{attribute 'linkalways'} 
{attribute 'no_explicit_call' := 'This FB is a CLASS and must be accessed using methods or properties'}
{attribute 'enable_dynamic_creation'}
FUNCTION_BLOCK Node_F_VN_InsertIntoContainer_SINT EXTENDS VisionNode
VAR
    nElement : _SINT(0);
    ipContainer : _ITcVnContainer;
    nIndex : _ULINT(0);
    hrPrev : _HRESULT(S_OK);
    hresult : _HRESULT(S_OK);
END_VAR

METHOD PUBLIC  Clone : I_Node
VAR
	pNode : POINTER TO Node_F_VN_InsertIntoContainer_SINT;
END_VAR
pNode := __NEW(Node_F_VN_InsertIntoContainer_SINT);
Clone := pNode^;
END_METHOD

METHOD FB_init : BOOL
VAR_INPUT
	bInitRetains : BOOL; // if TRUE, the retain variables are initialized (warm start / cold start)
	bInCopyCode : BOOL;  // if TRUE, the instance afterwards gets moved into the copy code (online change)
END_VAR
AddParameter('nElement', nElement);
AddInput('ipContainer', ipContainer);
AddParameter('nIndex', nIndex);
AddInput('hrPrev', hrPrev);
AddOutput('ipContainer', ipContainer);
AddOutput('hresult',hresult);
END_METHOD

METHOD PROTECTED OnExecute
hresult.Value := F_VN_InsertIntoContainer_SINT(
    nElement := nElement.Value,
    ipContainer := ipContainer.Value,
    nIndex := nIndex.Value,
    hrPrev:= hrPrev.Value);
END_METHOD

METHOD PUBLIC PreExecutionCheck
VAR_INPUT
	Check : I_PreExecutionChecks;
END_VAR
Check.IsTrue(ipContainer.IsValid, 'ipContainer must be a valid container');
Check.IsTrue(ipContainer.IsType(TC_GLOBAL_CONST_LIST.ContainerType_Vector_SINT), 'ipContainer contains incorrect type');
END_METHOD

END_FUNCTION_BLOCK

(* stored: Version 1.1.0.1, ProductVersion 3.1.4026.13
   POU Node_F_VN_InsertIntoContainer_SINT: Id {d080399f-bfbe-4776-aeff-af8e3fe8b050}, SpecialFunc None
   Folder Constructor: Id {1b5fda5a-fa5e-48be-b4e1-dbe204e4fdf0}
   Method Clone: Id {e8716c1e-3aac-42e3-9401-e12269070416}
   Method FB_init: Id {1bddfe7b-6452-4553-97e2-894aca56b2e8}
   Method OnExecute: Id {de629b7d-da56-4ea9-98b8-eef8813e93dd}
   Method PreExecutionCheck: Id {86dba2d6-d1bb-4d58-97e5-aac07615d96d} *)
